(* Logix 5000 project; controller CC100_EIPAdapter vendor 1 type 14 code 196 rev 32.14; software revision 32.03 *)

TASK MainTask (continuous, watchdog 500 ms) : MainProgram

MODULES
   Local : vendor 1 type 14 code 196 (5069 0, rev 32.14)
      RemoteIO_1A : vendor 1285 type 12 code 120 (Ethernet 192.168.50.113, rev 1.1, StandardDataDriven RPI 20 ms)
END_MODULES

VAR_GLOBAL   (* controller tags *)
   wAnalogInput : INT[2] := ([0] := 104, [1] := 112);
   wAnalogOutput : INT[2];
   wPTInput : INT[2] := ([0] := 3500, [1] := 3500);
   xDigitalOutput : INT;
   xDigtalInput : INT;
END_VAR

PROGRAM MainProgram   (* main routine MainRoutine *)

ROUTINE MainRoutine   (* ladder *)
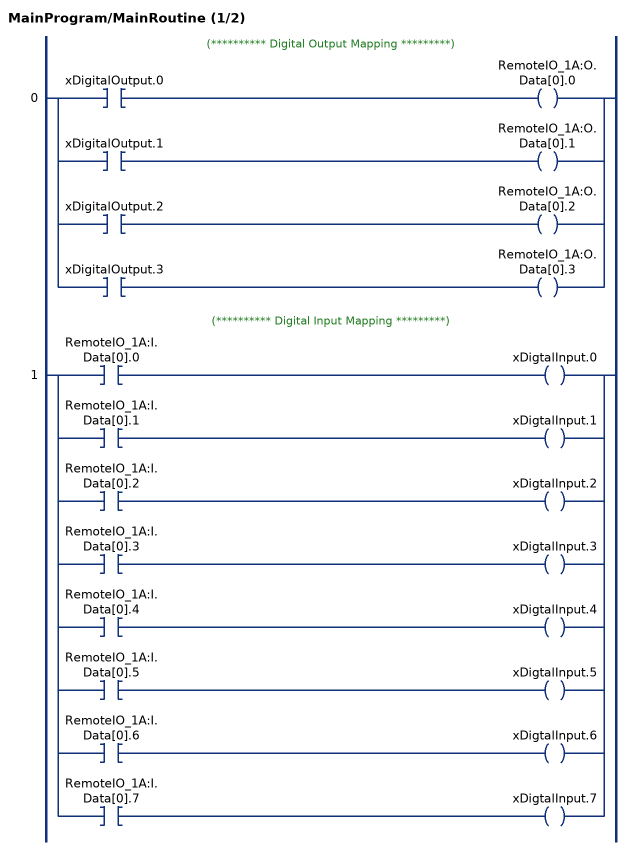
   // (********** Digital Output Mapping *********)
   0: [XIC(xDigitalOutput.0) OTE(RemoteIO_1A:O.Data[0].0) ,XIC(xDigitalOutput.1) OTE(RemoteIO_1A:O.Data[0].1) ,XIC(xDigitalOutput.2) OTE(RemoteIO_1A:O.Data[0].2) ,XIC(xDigitalOutput.3) OTE(RemoteIO_1A:O.Data[0].3) ];
   // (********** Digital Input Mapping *********)
   1: [XIC(RemoteIO_1A:I.Data[0].0) OTE(xDigtalInput.0) ,XIC(RemoteIO_1A:I.Data[0].1) OTE(xDigtalInput.1) ,XIC(RemoteIO_1A:I.Data[0].2) OTE(xDigtalInput.2) ,XIC(RemoteIO_1A:I.Data[0].3) OTE(xDigtalInput.3) ,XIC(RemoteIO_1A:I.Data[0].4) OTE(xDigtalInput.4) ,XIC(RemoteIO_1A:I.Data[0].5) OTE(xDigtalInput.5) ,XIC(RemoteIO_1A:I.Data[0].6) OTE(xDigtalInput.6) ,XIC(RemoteIO_1A:I.Data[0].7) OTE(xDigtalInput.7) ];
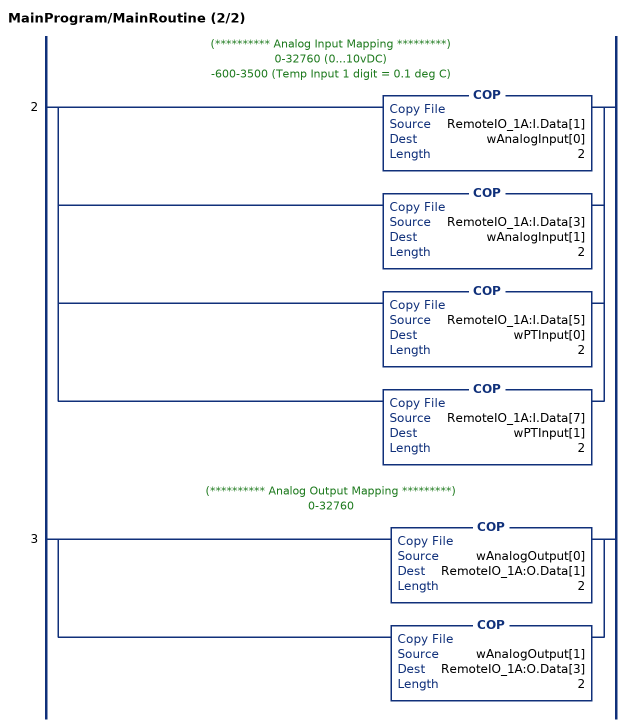
   // (********** Analog Input Mapping *********)
   // 0-32760 (0...10vDC)
   // -600-3500 (Temp Input 1 digit = 0.1 deg C)
   2: [[COP(RemoteIO_1A:I.Data[1],wAnalogInput[0],2) ,COP(RemoteIO_1A:I.Data[3],wAnalogInput[1],2) ] ,[COP(RemoteIO_1A:I.Data[5],wPTInput[0],2) ,COP(RemoteIO_1A:I.Data[7],wPTInput[1],2) ] ];
   // (********** Analog Output Mapping *********)
   // 0-32760
   3: [COP(wAnalogOutput[0],RemoteIO_1A:O.Data[1],2) ,COP(wAnalogOutput[1],RemoteIO_1A:O.Data[3],2) ];
END_ROUTINE
END_PROGRAM
